Staubli VAL3: findMove.pgx

program findMove(num x_nIndex, tool x_tTool, num& x_nMoveType[])
  local point l_pHere
  local num l_nResult
  local num l_nIndexTool
  local num l_nSize
  local num l_nMoveType
  local point l_pPoint[2]
  local joint l_jHere
  local bool l_bUnreach
begin
  //
  // MOVE TO THE POINT
  //
  // use the flange
  x_tTool=flange
  // get all the value that you need
  l_nSize=size(jEditPoint.tData)
  l_pHere=here(x_tTool,world)
  // get the point and the circle point
  call getPoint(l_pPoint,false,x_nIndex)
  pPoints[1].trsf=position(l_pPoint,world)
  pPoints[2].trsf={0,0,0,0,0,0}
  // Set to JOINT for default
  x_nMoveType=0
  // get the move TYPE
  call getMoveType(l_nMoveType,x_nIndex,false)
  //
  // move forward
  //
  if x_nIndex>0 and l_nMoveType==1
    // get the point and the circle point
    call getPoint(l_pPoint,false,x_nIndex-1)
    pPoints.trsf=position(l_pPoint,world)
    if distance(l_pHere,pPoints)<25
      // set to linear
      x_nMoveType=1
    elseIf setFrame(pPoints,pPoints[1],pPoints[2],fSetFrame)==0
      // check frame
      l_pHere=here(x_tTool,fSetFrame)
      pPoints[1].trsf=position(pPoints[1],fSetFrame)
      if l_pHere.trsf.x>=0 and l_pHere.trsf.x<=pPoints[1].trsf.x and abs(l_pHere.trsf.y)<10 and abs(l_pHere.trsf.z)<10
        // set to linear
        x_nMoveType=1
      endIf
    endIf
  endIf
  //
  // move back
  //
  if x_nIndex<(l_nSize-1) and x_nMoveType!=1
    call getMoveType(l_nMoveType,x_nIndex+1,false)
    if l_nMoveType==1
      // get the point and the circle point
      call getPoint(l_pPoint,false,x_nIndex)
      pPoints[1].trsf=position(l_pPoint,world)
      // get the point and the circle point
      call getPoint(l_pPoint,false,x_nIndex+1)
      pPoints.trsf=position(l_pPoint,world)
      if distance(l_pHere,pPoints)<25
        // switch to linear
        x_nMoveType=1
      elseIf setFrame(pPoints,pPoints[1],pPoints[2],fSetFrame)==0
        // check frame
        l_pHere=here(x_tTool,fSetFrame)
        pPoints[1].trsf=position(pPoints[1],fSetFrame)
        if l_pHere.trsf.x>=0 and l_pHere.trsf.x<=pPoints[1].trsf.x and abs(l_pHere.trsf.y)<10 and abs(l_pHere.trsf.z)<10
          // set to linear
          x_nMoveType=1
        endIf
      endIf
    endIf
  endIf
end
